// TwinCAT 3 PLC project BufferModeV2
// ProgramVersion: 3.1.4024.0
// libraries:
//   Tc2_MC2, * (Beckhoff Automation GmbH)
//   Tc2_Standard, * (Beckhoff Automation GmbH)
//   Tc2_System, * (Beckhoff Automation GmbH)
//   Tc3_Module, * (Beckhoff Automation GmbH)
// project tree:
//   / PlcTask.TcTTO
//   POUs/ MAIN.TcPOU
// real-time tasks:
//   TASK PlcTask: cycle T#10ms, priority 20, ADS port 350
// motion (NC):
//   TASK NC-Task 1 SAF: cycle T#2ms, priority 4, ADS port 501
//   TASK NC-Task 1 SVB: cycle T#10ms, priority 8, ADS port 511
//   AXIS Axis 1 (id 1)
//     OtherSettings: AllowMotionCmdToSlave=true
//     encoder EncType=1
//     drive DrvType=5
//       Analog: TorqueSetpointScale=10, ScaleFactorActTorque=0.1
//       TimeComp: TaskDelayCycles=1
//     controller CtrType=1
//       CtrPara: PriorControlFactor=1
//         Observer: BandWidth=20
// variable links:
//   BufferModeV2/BufferModeV2 Instance <-> NC-Task 1 SAF/Axes/Axis 1
//     PlcTask Inputs/MAIN.Axis_1.NcToPlc <-> Outputs/ToPlc
//     PlcTask Outputs/MAIN.Axis_1.PlcToNc <-> Inputs/FromPlc

CONFIGURATION BufferModeV2
    RESOURCE PLC ON TwinCAT3
        TASK PlcTask(INTERVAL := T#10ms, PRIORITY := 20);
        PROGRAM MAIN WITH PlcTask : MAIN;
    END_RESOURCE
END_CONFIGURATION

// ---- POUs/MAIN.TcPOU
PROGRAM MAIN
VAR
	Axis_1 			: AXIS_REF;
	fbPowerOn 		: MC_Power;
	fbMoveAbs 		: MC_MoveAbsolute;
	fbMoveAbs2 		: MC_MoveAbsolute;
	fbMoveRel 		: MC_MoveRelative;
	fbMoveRel2 		: MC_MoveRelative;

	
	mcBufferMode : MC_BufferMode;
	bGotoPos1: BOOL := FALSE;
	eMovePos : (E_Init, E_POS1,  E_POS2, E_POS3,E_POS4) := E_init;
	bEnableAxis: BOOL;
END_VAR

fbPowerOn(Axis:= Axis_1, Enable:= bEnableAxis, Enable_Positive:=bEnableAxis, Enable_Negative:= bEnableAxis);

IF bGotoPos1 THEN
	eMovePos := E_POS1;
END_IF
CASE eMovePos OF
	E_init:
		fbMoveAbs(Axis:= Axis_1, Execute:= FALSE);
		fbMoveRel(Axis:= Axis_1, Execute:= FALSE);
	E_POS1:
		fbMoveAbs(Axis:= Axis_1, Execute:= bGotoPos1, Position:= 200, Velocity:= 15, Acceleration:= 10, Deceleration:= 10, BufferMode:= MC_Buffered );
		IF fbMoveAbs.Busy THEN
			fbMoveAbs(Axis:= Axis_1, Execute:= FALSE);
			bGotoPos1 := FALSE;
			eMovePos := E_POS2;
		END_IF
	
	E_POS2:
		fbMoveRel(Axis:= Axis_1, Execute:= TRUE, Distance:= 550, Velocity:= 55, Acceleration:= 15, Deceleration:= 15, BufferMode:= MC_Aborting );
		IF fbMoveRel.Active THEN
			fbMoveRel(Axis:= Axis_1, Execute:= FALSE);
			eMovePos := E_POS3;
		END_IF
		
	E_POS3:
	fbMoveRel2(Axis:= Axis_1, Execute:= TRUE, Distance:= 550, Velocity:= 80, Acceleration:= 15, Deceleration:= 15, BufferMode:= MC_Buffered );
		IF fbMoveRel2.Active THEN
			fbMoveRel2(Axis:= Axis_1, Execute:= FALSE);
			eMovePos := E_POS4;
		END_IF
	E_POS4:
	fbMoveAbs2(Axis:= Axis_1, Execute:= TRUE, Position:= 0, Velocity:= 300, Acceleration:= 10, Deceleration:= 10, BufferMode:= MC_Buffered );
		IF fbMoveAbs2.Active THEN
			fbMoveAbs2(Axis:= Axis_1, Execute:= FALSE);
			eMovePos := E_Init;
		END_IF
		
END_CASE

END_PROGRAM
